Yaskawa INFORM job: OK_R2_O6-7(-90,0)OKKR.JBI

/JOB
//NAME OK_R2_O6-7(-90,0)OKKR
///FOLDERNAME X4
//POS
///NPOS 133,133,131,6,0,0
///TOOL 0
///POSTYPE PULSE
///PULSE
C00000=60285,-10095,-87170,10907,88181,-3199
C00001=89581,-19308,-95624,3409,86568,14234
C00002=122268,-16957,-60346,12820,63530,51265
C00003=120644,-15828,-53256,21467,67230,40646
C00004=120644,-14098,-51953,21456,67311,40660
C00005=120643,-14518,-52071,21476,67179,40636
C00006=120643,-15104,-51195,21601,66394,40485
C00007=120642,-17255,-54944,21425,67517,40699
C00008=120642,-17255,-54944,21425,67517,40699
C00009=124252,-5529,-45197,19318,66732,41820
C00010=124248,-5319,-45028,19320,66737,41819
C00011=124218,-3848,-43837,19334,66766,41814
C00012=124229,-4373,-44263,19329,66756,41816
C00013=124229,-5024,-43316,19456,65890,41667
C00014=124282,-6279,-47079,19198,67460,41953
C00015=120646,-13302,-53858,21234,68787,40941
C00016=120646,-14762,-51940,21506,66983,40600
C00017=120646,-14720,-50898,21598,66406,40487
C00018=120830,-17522,-52800,21535,66110,40497
C00019=120651,-14728,-51994,21496,67029,40610
C00020=120646,-14787,-50945,21602,66406,40490
C00021=120646,-14870,-50970,21605,66385,40483
C00022=120646,-14919,-51008,21604,66373,40480
C00023=120646,-15018,-51986,21521,66887,40581
C00024=120646,-13567,-53912,21247,68691,40923
C00025=105915,-38442,-90635,28282,81378,38856
C00026=57484,-69477,-110718,42573,54444,32820
C00027=-3643,-76224,-106676,-19950,71810,-76872
C00028=36671,-135259,-121545,10452,42336,6075
C00029=153552,-182601,-115262,-69180,49813,-17515
C00030=130897,-39590,-67652,-38094,64357,-42352
C00031=133939,-4658,-36155,-42635,61093,-39682
C00032=121252,36500,14973,-37087,50890,-41500
C00033=120918,45177,26978,-38391,48402,-40561
C00034=121382,52420,34740,-38113,53329,-33841
C00035=121382,52654,36258,-38487,52687,-33558
C00036=121382,52420,34740,-38113,53329,-33841
C00037=121377,54820,37402,-38294,53006,-33703
C00038=121382,52420,34740,-38113,53329,-33841
C00039=121917,44386,26656,-39102,48682,-40133
C00040=134879,58255,40786,-46614,53825,-35408
C00041=134959,60833,45092,-47358,52948,-34841
C00042=134959,61144,46552,-47770,52438,-34533
C00043=134959,60875,45298,-47416,52875,-34797
C00044=134857,63056,47803,-47604,52533,-34650
C00045=134959,60875,45298,-47416,52875,-34797
C00046=132891,53596,35323,-45210,53491,-36376
C00047=128554,62524,39730,-40860,62650,-37664
C00048=124660,52481,28282,-31369,57719,-36489
C00049=124396,62029,43751,-32872,53681,-35247
C00050=124397,61721,41951,-32506,54487,-35529
C00051=124441,58589,39965,-32677,54175,-35400
C00052=133765,73788,57651,-38360,55527,-31292
C00053=134326,62719,39703,-36596,60072,-32844
C00054=135410,51148,31829,-38776,48591,-44747
C00055=138156,57586,38014,-40647,49456,-43620
C00056=137577,66731,52697,-42929,45898,-42064
C00057=133639,60157,45125,-39794,45011,-44001
C00058=132456,59443,46653,-39908,43454,-43903
C00059=132752,49719,31225,-37339,47144,-45563
C00060=132976,-10381,-34918,-42251,48570,-38774
C00061=134698,-65118,-78640,-42103,61094,-39224
C00062=147917,-167168,-112708,-64264,48960,-21968
C00063=119754,-187210,-115895,-71836,42621,-17929
C00064=119758,-186866,-115850,-71681,42673,-18021
C00065=53896,-172979,-113746,-63904,34565,-25257
C00066=23682,-170517,-113316,-58323,27834,-29716
C00067=-3643,-76224,-106676,-19950,71810,-76872
C00068=64381,-28256,-98450,-10969,86693,-48952
C00069=88971,-14667,-95667,-7498,68279,-41414
C00070=119588,-13110,-62704,-15013,73832,-42943
C00071=119588,-13110,-62704,-15013,73832,-42943
C00072=120558,-12095,-59649,-15670,72677,-42495
C00073=120559,-10147,-58145,-15666,72751,-42503
C00074=120558,-10769,-58628,-15667,72729,-42501
C00075=120558,-10769,-58628,-15667,72729,-42501
C00076=120558,-11635,-57914,-15738,71876,-42387
C00077=120555,-12891,-60896,-15641,73024,-42540
C00078=95040,4780,-47974,-473,71962,-50162
C00079=96326,6971,-43876,-1258,70580,-49764
C00080=96504,8188,-42807,-1365,70550,-49710
C00081=96432,7698,-43239,-1322,70563,-49732
C00082=96432,6895,-42576,-1327,69744,-49725
C00083=96090,5943,-45717,-1110,71182,-49845
C00084=120646,-13948,-53489,-21604,68017,-40999
C00085=120646,-15353,-51537,-21891,66225,-40651
C00086=120646,-15164,-50572,-21969,65764,-40561
C00087=120651,-15325,-51597,-21886,66274,-40659
C00088=120458,-18091,-52377,-21925,65351,-40547
C00089=120646,-15383,-50573,-21989,65664,-40541
C00090=120646,-15549,-50757,-21980,65686,-40545
C00091=120646,-15089,-51509,-21872,66335,-40673
C00092=120646,-13673,-53452,-21587,68128,-41020
C00093=109799,-58506,-103025,-1655,56640,-68945
C00094=72582,-82093,-114007,4014,51361,-71324
C00095=52067,-53786,-27019,64889,38361,-39682
C00096=120741,-100002,-85602,9981,27010,44029
C00097=119621,-44404,-59771,8419,41423,45013
C00098=117663,-2811,-38597,8399,52217,45191
C00099=120702,21452,-13699,5381,57938,46744
C00100=116335,56883,35867,37385,59322,29596
C00101=116196,48699,28248,37279,59768,29706
C00102=116239,51251,31028,37399,59426,29593
C00103=116211,49643,29272,37323,59642,29665
C00104=116211,49822,31006,37666,58859,29354
C00105=116172,47372,26030,37059,60326,29912
C00106=106186,56602,32458,40868,65398,27238
C00107=106572,58996,37080,41208,63985,26816
C00108=106692,61436,39855,41307,63581,26700
C00109=106591,59390,37526,41224,63919,26799
C00110=106591,59599,39424,41561,63110,26445
C00111=106493,57459,35257,41134,64272,26904
C00112=115846,42546,19421,36690,61750,30302
C00113=117555,46608,31297,40428,52454,27269
C00114=120687,94317,83744,31652,39524,45736
C00115=120569,90994,80772,31662,39672,45727
C00116=110051,72582,62222,48229,50609,21848
C00117=111679,66904,55317,43745,47468,25399
C00118=112458,62952,41455,33837,55853,32000
C00119=111893,69063,52340,37068,50562,29781
C00120=111570,73580,54354,35260,54156,30929
C00121=111490,70901,52297,35345,54097,30866
C00122=107052,75469,60535,41045,50946,27156
C00123=107111,76128,56911,37464,55825,29367
C00124=111954,67372,45051,34070,56101,31848
C00125=111993,73411,55309,35316,53423,30857
C00126=113179,72507,56659,35287,51867,30842
C00127=112397,61419,38958,33599,56505,32200
C00128=120702,23915,-11347,5391,57756,46734
C00129=120707,-6637,-31564,7607,37304,45295
C00130=120737,-64904,-74687,7327,38208,45433
C00131=93974,-150495,-124706,8327,75713,42563
C00132=8894,-114644,-114160,10000,88881,39323
BC00000=260410,492998,972848
BC00001=270030,483686,999233
BC00002=258993,456898,1075139
BC00003=256299,434832,1075139
BC00004=256299,434832,1075139
BC00005=256299,434832,1075139
BC00006=256299,434832,1075139
BC00007=256299,434832,1075139
BC00008=203965,434832,1075139
BC00009=203965,434832,1075139
BC00010=203965,434832,1075139
BC00011=203965,434832,1075139
BC00012=203965,434832,1075139
BC00013=203965,434832,1075139
BC00014=203965,434832,1075139
BC00015=255837,442462,1075139
BC00016=256167,437012,1075139
BC00017=256299,434832,1075139
BC00018=256299,434832,1075139
BC00019=256299,434832,1075139
BC00020=251596,434014,1075139
BC00021=199069,424971,1075139
BC00022=194363,424171,1075139
BC00023=194231,426350,1075139
BC00024=193901,431800,1075139
BC00025=193901,431800,1075139
BC00026=193901,502169,1075139
BC00027=199448,515539,1075137
BC00028=185032,493226,660827
BC00029=170886,507346,17
BC00030=170886,499137,17
BC00031=170886,500820,17
BC00032=170886,503207,17
BC00033=170886,506149,17
BC00034=170886,504467,17
BC00035=170886,504467,17
BC00036=170886,504467,17
BC00037=170886,504467,17
BC00038=170886,504467,17
BC00039=170886,505099,17
BC00040=170886,505099,17
BC00041=170886,505099,17
BC00042=170886,505099,17
BC00043=170886,505099,17
BC00044=170886,505099,17
BC00045=170886,505099,17
BC00046=170886,505099,17
BC00047=183787,509866,15
BC00048=183787,509866,15
BC00049=183787,509866,15
BC00050=183787,509866,15
BC00051=183787,509866,15
BC00052=183787,509866,15
BC00053=183787,509866,15
BC00054=183787,509866,15
BC00055=183787,509866,15
BC00056=183787,509866,15
BC00057=183787,509866,15
BC00058=183787,509866,15
BC00059=183787,509866,15
BC00060=170886,507200,17
BC00061=170886,511894,17
BC00062=170886,502226,17
BC00063=170886,505869,17
BC00064=170886,506079,17
BC00065=170886,509232,17
BC00066=170886,502507,17
BC00067=199448,515539,1075137
BC00068=143041,501148,792030
BC00069=138642,496819,917141
BC00070=200892,451069,1075139
BC00071=195544,434280,1021239
BC00072=195544,434280,1021238
BC00073=195544,434280,1021238
BC00074=195544,434280,1021238
BC00075=195544,434280,1021238
BC00076=195544,434280,1021238
BC00077=195544,434280,1021238
BC00078=195544,434280,1021238
BC00079=195544,434280,1021238
BC00080=195544,434280,1021238
BC00081=195544,434280,1021238
BC00082=195544,434280,1021238
BC00083=195544,434280,1021238
BC00084=186560,442338,1075139
BC00085=186271,436877,1075139
BC00086=186156,434693,1075139
BC00087=186156,434693,1075139
BC00088=186156,434693,1075139
BC00089=243368,424735,1075139
BC00090=248072,423926,1075139
BC00091=248187,426110,1075139
BC00092=248476,431571,1075139
BC00093=248476,431571,1075139
BC00094=154886,508880,1075139
BC00095=226129,512135,483138
BC00096=268409,479745,74497
BC00097=268409,503413,53619
BC00098=268409,500913,17
BC00099=268409,507760,17
BC00100=268944,502290,17
BC00101=268944,493646,17
BC00102=268944,493646,17
BC00103=268944,493646,17
BC00104=268944,493646,17
BC00105=268944,493646,17
BC00106=268944,493646,17
BC00107=268944,493646,17
BC00108=268944,493646,17
BC00109=268944,493646,17
BC00110=268944,493646,17
BC00111=268944,493646,17
BC00112=268944,491895,17
BC00113=268943,496238,12
BC00114=254289,537584,17
BC00115=254289,537584,17
BC00116=268943,512909,14
BC00117=268944,512909,12
BC00118=268943,512909,14
BC00119=268943,512909,12
BC00120=268943,512909,12
BC00121=268943,512909,12
BC00122=268943,512909,14
BC00123=268943,512909,14
BC00124=268943,512909,14
BC00125=268943,512909,14
BC00126=268943,512909,14
BC00127=268943,512909,14
BC00128=268409,510422,17
BC00129=268409,508881,17
BC00130=268409,508951,17
BC00131=268409,511824,17
BC00132=268409,511683,17
EC00000=798297,-183828
EC00001=798261,-183829
EC00002=798156,-183832
EC00003=798156,-183832
EC00004=798156,-183832
EC00005=798156,-183832
EC00006=798156,-183832
EC00007=798156,-183832
EC00008=798156,-183832
EC00009=798156,-183832
EC00010=798156,-183832
EC00011=798156,-183832
EC00012=798156,-183832
EC00013=798156,-183832
EC00014=798156,-183832
EC00015=798156,-183832
EC00016=798156,-183832
EC00017=798156,-183832
EC00018=798156,-183832
EC00019=798156,-183832
EC00020=798156,-183832
EC00021=798156,-183832
EC00022=798156,-183832
EC00023=798156,-183832
EC00024=798156,-183832
EC00025=798156,-183832
EC00026=798156,-183832
EC00027=798156,-183832
EC00028=798156,-183832
EC00029=798156,-183832
EC00030=798156,-183832
EC00031=798156,-183832
EC00032=798156,-183832
EC00033=798156,-183832
EC00034=798156,-183832
EC00035=798156,-183832
EC00036=798156,-183832
EC00037=798156,-183832
EC00038=798156,-183832
EC00039=798156,-183832
EC00040=798156,-183832
EC00041=798156,-183832
EC00042=798156,-183832
EC00043=798156,-183832
EC00044=798156,-183832
EC00045=798156,-183832
EC00046=798156,-183832
EC00047=798154,-183831
EC00048=798154,-183831
EC00049=798154,-183831
EC00050=798154,-183831
EC00051=798154,-183831
EC00052=798154,-183831
EC00053=798154,-183831
EC00054=798154,-183831
EC00055=798154,-183831
EC00056=798154,-183831
EC00057=798154,-183831
EC00058=798154,-183831
EC00059=798154,-183831
EC00060=798156,-183832
EC00061=798156,-183832
EC00062=798156,-183832
EC00063=867082,-372677
EC00064=885768,-557346
EC00065=906795,-866627
EC00066=886351,-984978
EC00067=798156,-1296783
EC00068=798156,-1296783
EC00069=798156,-1296783
EC00070=798156,-1296783
EC00071=798156,-1296783
EC00072=798154,-1296783
EC00073=798154,-1296783
EC00074=798154,-1296783
EC00075=798154,-1296783
EC00076=798154,-1296783
EC00077=798154,-1296783
EC00078=798154,-1296783
EC00079=798154,-1296783
EC00080=798154,-1296783
EC00081=798154,-1296783
EC00082=798154,-1296783
EC00083=798154,-1296783
EC00084=798156,-1296783
EC00085=798156,-1296783
EC00086=798156,-1296783
EC00087=798156,-1296783
EC00088=798156,-1296783
EC00089=798156,-1296783
EC00090=798156,-1296783
EC00091=798156,-1296783
EC00092=798156,-1296783
EC00093=798156,-1296783
EC00094=798156,-1296783
EC00095=798156,-1296783
EC00096=798156,-1296783
EC00097=798156,-1296783
EC00098=798156,-1296783
EC00099=798156,-1296783
EC00100=798156,-1296783
EC00101=798156,-1296783
EC00102=798156,-1296783
EC00103=798156,-1296783
EC00104=798156,-1296783
EC00105=798156,-1296783
EC00106=798156,-1296783
EC00107=798156,-1296783
EC00108=798156,-1296783
EC00109=798156,-1296783
EC00110=798156,-1296783
EC00111=798156,-1296783
EC00112=798156,-1296783
EC00113=798154,-1296785
EC00114=798156,-1296783
EC00115=798156,-1296783
EC00116=798155,-1296784
EC00117=798154,-1296784
EC00118=798155,-1296784
EC00119=798154,-1296784
EC00120=798155,-1296784
EC00121=798155,-1296784
EC00122=798155,-1296784
EC00123=798155,-1296784
EC00124=798155,-1296784
EC00125=798155,-1296784
EC00126=798156,-1296783
EC00127=798156,-1296783
EC00128=798156,-1296783
EC00129=798156,-1296783
EC00130=798156,-1296783
///POSTYPE BASE
///RECTAN
///RCONF 0,0,0,0,1,0,0,0,0,0,0,0,0,0,0,0,0,0,0,0,0,0,0,0
P00006=2.006,1.622,-0.565,0.0000,0.0000,0.0000
P00021=0.073,2.058,-0.109,0.0000,0.0000,0.0000
P00022=2.006,1.622,-0.565,0.0000,0.0000,0.0000
///RCONF 0,0,0,0,0,0,0,0,0,0,0,0,0,0,0,0,0,0,0,0,0,0,0,0
P00023=-2.957,-4.083,2.762,0.0000,0.0000,0.0000
P00025=3.643,0.007,-2.585,0.0000,0.0000,0.0000
P00026=2.644,0.055,-2.583,0.0000,0.0000,0.0000
//INST
///DATE 2024/11/13 18:37
///ATTR SC,RW
///GROUP1 RB1,BS1
///GROUP2 ST1
NOP
'OK_r2_O6-7(-90,0)
'Spoina W6
'Path S1006
MOVJ C00000 BC00000 VJ=100.00  +MOVJ EC00000 VJ=10.00
MOVJ C00001 BC00001 VJ=100.00  +MOVJ EC00001 VJ=10.00
SFTOF3D
MOVJ C00002 BC00002 VJ=100.00  +MOVJ EC00002 VJ=100.00
SMOVL C00003 BC00003 V=100.0  +MOVJ EC00003
SREFP 3 C00004 BC00004  +REFP EC00004
CALL JOB:SEARCH-R1-S13D
SET P021 P006
SFTON3D P021
SMOVL C00005 BC00005 V=100.0  +MOVJ EC00005
SREFP 3 C00006 BC00006  +REFP EC00006
CALL JOB:SEARCH-R1-S13D
SET P021 P006
SFTON3D P021
SMOVL C00007 BC00007 V=100.0  +MOVJ EC00007
MOVL C00008 BC00008 V=400.0  +MOVJ EC00008 VJ=100.00
MOVL C00009 BC00009 V=400.0  +MOVJ EC00009 VJ=100.00
SMOVL C00010 BC00010 V=100.0  +MOVJ EC00010
SREFP 3 C00011 BC00011  +REFP EC00011
CALL JOB:SEARCH-R1-S13D
SET P022 P006
SFTON3D P022
SMOVL C00012 BC00012 V=100.0  +MOVJ EC00012
SREFP 3 C00013 BC00013  +REFP EC00013
CALL JOB:SEARCH-R1-S13D
SET P022 P006
SFTON3D P022
SMOVL C00014 BC00014 V=100.0  +MOVJ EC00014
'Path W937
SFTOF3D
MOVJ C00015 BC00015 VJ=50.00  +MOVJ EC00015 VJ=100.00
SMOVL C00016 BC00016 V=400.0  +MOVJ EC00016
SFTON3D P021
SMOVL C00017 BC00017 V=100.0 PL=0  +MOVJ EC00017
SREFP 1 C00018 BC00018  +REFP EC00018
SREFP 2 C00019 BC00019  +REFP EC00019
MACRO1 MJ#(0) ARGF6
ARCON
SMOVL C00020 BC00020 V=8.3  +MOVJ EC00020
SFTON3D P022
SMOVL C00021 BC00021 V=8.3  +MOVJ EC00021
SMOVL C00022 BC00022 V=8.3  +MOVJ EC00022
ARCOF
SMOVL C00023 BC00023 V=400.0  +MOVJ EC00023
SFTOF3D
SMOVL C00024 BC00024 V=1000.0  +MOVJ EC00024
MOVJ C00025 BC00025 VJ=100.00  +MOVJ EC00025 VJ=10.00
MOVJ C00026 BC00026 VJ=100.00  +MOVJ EC00026 VJ=100.00
MOVJ C00027 BC00027 VJ=100.00  +MOVJ EC00027 VJ=100.00
SFTOF3D
CALL JOB:CLEAN-R1_KM_NEW
'wire_cut
SFTOF
'wire_cut
MOVJ C00028 BC00028 VJ=100.00  +MOVJ EC00028 VJ=100.00
MOVJ C00029 BC00029 VJ=100.00  +MOVJ EC00029 VJ=100.00
MOVJ C00030 BC00030 VJ=50.00  +MOVJ EC00030 VJ=100.00
MOVJ C00031 BC00031 VJ=50.00  +MOVJ EC00031 VJ=100.00
'Path S1300
SFTOF3D
MOVJ C00032 BC00032 VJ=50.00  +MOVJ EC00032 VJ=100.00
MOVL C00033 BC00033 V=100.0  +MOVJ EC00033 VJ=100.00
SMOVL C00034 BC00034 V=100.0  +MOVJ EC00034
SREFP 3 C00035 BC00035  +REFP EC00035
CALL JOB:SEARCH-R1-S13D
SET P025 P006
SFTON3D P025
SMOVL C00036 BC00036 V=100.0  +MOVJ EC00036
SREFP 3 C00037 BC00037  +REFP EC00037
CALL JOB:SEARCH-R1-S13D
SET P025 P006
SFTON3D P025
SMOVL C00038 BC00038 V=100.0  +MOVJ EC00038
MOVL C00039 BC00039 V=400.0  +MOVJ EC00039 VJ=100.00
SMOVL C00040 BC00040 V=400.0  +MOVJ EC00040
SMOVL C00041 BC00041 V=100.0  +MOVJ EC00041
SREFP 3 C00042 BC00042  +REFP EC00042
CALL JOB:SEARCH-R1-S13D
SET P026 P006
SFTON3D P026
SMOVL C00043 BC00043 V=100.0  +MOVJ EC00043
SREFP 3 C00044 BC00044  +REFP EC00044
CALL JOB:SEARCH-R1-S13D
SET P026 P006
SFTON3D P026
SMOVL C00045 BC00045 V=100.0  +MOVJ EC00045
MOVL C00046 BC00046 V=1000.0  +MOVJ EC00046 VJ=100.00
'Path W1301
SFTOF3D
SFTON3D P025
MOVJ C00047 BC00047 VJ=50.00  +MOVJ EC00047 VJ=100.00
SMOVL C00048 BC00048 V=400.0  +MOVJ EC00048
SFTON3D P025
SMOVL C00049 BC00049 V=100.0 PL=0  +MOVJ EC00049
SREFP 1 C00050 BC00050  +REFP EC00050
SREFP 2 C00051 BC00051  +REFP EC00051
MACRO1 MJ#(0) ARGF6
ARCON
SWVON WEV#(30)
SMOVL C00052 BC00052 V=8.3  +MOVJ EC00052
ARCOF
SWVOF
MOVJ C00053 BC00053 VJ=50.00  +MOVJ EC00053 VJ=10.00
SFTOF3D
MOVJ C00054 BC00054 VJ=50.00  +MOVJ EC00054 VJ=10.00
MOVJ C00055 BC00055 VJ=50.00  +MOVJ EC00055 VJ=10.00
MACRO1 MJ#(0) ARGF6
SFTON3D P026
SMOVL C00056 BC00056 V=100.0  +MOVJ EC00056
ARCON
SWVON WEV#(30)
ARCON
SMOVL C00057 BC00057 V=7.5  +MOVJ EC00057
SMOVL C00058 BC00058 V=10.0  +MOVJ EC00058
ARCOF
SWVOF
MOVJ C00059 BC00059 VJ=100.00  +MOVJ EC00059 VJ=10.00
SFTOF3D
MOVJ C00060 BC00060 VJ=100.00  +MOVJ EC00060 VJ=100.00
MOVJ C00061 BC00061 VJ=100.00  +MOVJ EC00061 VJ=100.00
'OBROT_SPRAWDZIC
MOVJ C00062 BC00062 VJ=100.00  +MOVJ EC00062 VJ=100.00
MOVJ C00063 BC00063 VJ=100.00  +MOVJ EC00063 VJ=100.00
MOVJ C00064 BC00064 VJ=100.00  +MOVJ EC00064 VJ=100.00
MOVJ C00065 BC00065 VJ=100.00  +MOVJ EC00065 VJ=100.00
MOVJ C00066 BC00066 VJ=100.00  +MOVJ EC00066 VJ=100.00
MOVJ C00067 BC00067 VJ=100.00  +MOVJ EC00067 VJ=100.00
CALL JOB:CLEAN-R1_KM_NEW
'wire_cut
'wire_cut
'Path S1296
MOVJ C00068 BC00068 VJ=100.00  +MOVJ EC00068 VJ=10.00
MOVJ C00069 BC00069 VJ=100.00  +MOVJ EC00069 VJ=10.00
SFTOF3D
MOVJ C00070 BC00070 VJ=100.00  +MOVJ EC00070 VJ=100.00
MOVL C00071 BC00071 V=100.0  +MOVJ EC00071 VJ=100.00
SMOVL C00072 BC00072 V=100.0  +MOVJ EC00072
SREFP 3 C00073 BC00073  +REFP EC00073
CALL JOB:SEARCH-R1-S13D
SET P021 P006
SFTON3D P021
SMOVL C00074 BC00074 V=100.0  +MOVJ EC00074
SMOVL C00075 BC00075 V=100.0  +MOVJ EC00075
SREFP 3 C00076 BC00076  +REFP EC00076
CALL JOB:SEARCH-R1-S13D
SET P021 P006
SFTON3D P021
SFTOF3D
SMOVL C00077 BC00077 V=100.0  +MOVJ EC00077
MOVJ C00078 BC00078 VJ=50.00  +MOVJ EC00078 VJ=50.00
'POMIAR 2
SMOVL C00079 BC00079 V=100.0  +MOVJ EC00079
SREFP 3 C00080 BC00080  +REFP EC00080
CALL JOB:SEARCH-R1-S13D
SET P022 P006
SFTON3D P022
SMOVL C00081 BC00081 V=100.0  +MOVJ EC00081
SREFP 3 C00082 BC00082  +REFP EC00082
CALL JOB:SEARCH-R1-S13D
SET P022 P006
SFTON3D P022
SMOVL C00083 BC00083 V=100.0  +MOVJ EC00083
'Path W1297
SFTOF3D
SFTON3D P021
MOVJ C00084 BC00084 VJ=50.00  +MOVJ EC00084 VJ=100.00
SMOVL C00085 BC00085 V=400.0  +MOVJ EC00085
SMOVL C00086 BC00086 V=100.0 PL=0  +MOVJ EC00086
SREFP 1 C00087 BC00087  +REFP EC00087
SREFP 2 C00088 BC00088  +REFP EC00088
MACRO1 MJ#(0) ARGF6
ARCON
SMOVL C00089 BC00089 V=9.2  +MOVJ EC00089
SMOVL C00090 BC00090 V=9.2  +MOVJ EC00090
ARCOF
SWVOF
SMOVL C00091 BC00091 V=400.0  +MOVJ EC00091
SMOVL C00092 BC00092 V=1000.0  +MOVJ EC00092
MOVJ C00093 BC00093 VJ=100.00  +MOVJ EC00093 VJ=10.00
MOVJ C00094 BC00094 VJ=100.00  +MOVJ EC00094 VJ=10.00
SFTOF3D
CALL JOB:CLEAN-R1_KM_NEW
'wire_cut
'wire_cut
'Spoina W7
MOVJ C00095 BC00095 VJ=100.00  +MOVJ EC00095 VJ=10.00
MOVJ C00096 BC00096 VJ=100.00  +MOVJ EC00096 VJ=100.00
MOVJ C00097 BC00097 VJ=100.00  +MOVJ EC00097 VJ=50.00
MOVJ C00098 BC00098 VJ=100.00  +MOVJ EC00098 VJ=10.00
MOVJ C00099 BC00099 VJ=100.00  +MOVJ EC00099 VJ=100.00
'Path S1298
SFTOF3D
MOVL C00100 BC00100 V=400.0  +MOVJ EC00100 VJ=100.00
SMOVL C00101 BC00101 V=100.0  +MOVJ EC00101
SREFP 3 C00102 BC00102  +REFP EC00102
CALL JOB:SEARCH-R1-S13D
SET P023 P006
SFTON3D P023
SMOVL C00103 BC00103 V=100.0  +MOVJ EC00103
SREFP 3 C00104 BC00104  +REFP EC00104
CALL JOB:SEARCH-R1-S13D
SET P023 P006
SFTON3D P023
SFTOF3D
SMOVL C00105 BC00105 V=100.0  +MOVJ EC00105
'POMIAR 2
MOVJ C00106 BC00106 VJ=50.00  +MOVJ EC00106 VJ=50.00
SMOVL C00107 BC00107 V=100.0  +MOVJ EC00107
SREFP 3 C00108 BC00108  +REFP EC00108
CALL JOB:SEARCH-R1-S13D
SET P021 P006
SFTON3D P021
SMOVL C00109 BC00109 V=100.0  +MOVJ EC00109
SREFP 3 C00110 BC00110  +REFP EC00110
CALL JOB:SEARCH-R1-S13D
SET P021 P006
SFTON3D P021
SMOVL C00111 BC00111 V=166.7  +MOVJ EC00111
MOVL C00112 BC00112 V=400.0  +MOVJ EC00112 VJ=100.00
'Path W1299
SFTOF3D
SFTON3D P023
SMOVL C00113 BC00113 V=100.0 PL=0  +MOVJ EC00113
SREFP 1 C00114 BC00114  +REFP EC00114
SREFP 2 C00115 BC00115  +REFP EC00115
MACRO1 MJ#(0) ARGF14
ARCON
SWVON WEV#(30)
SMOVL C00116 BC00116 V=9.2  +MOVJ EC00116
SMOVL C00117 BC00117 V=9.2  +MOVJ EC00117
ARCOF
SWVOF
MOVJ C00118 BC00118 VJ=100.00  +MOVJ EC00118 VJ=10.00
SFTON3D P021
SMOVL C00119 BC00119 V=100.0 PL=0  +MOVJ EC00119
REFP 1 RB1 C00120 BC00120
REFP 2 RB1 C00121 BC00121
ARCON
SWVON WEV#(30)
SMOVL C00122 BC00122 V=7.5  +MOVJ EC00120
ARCOF
SWVOF
MOVJ C00123 BC00123 VJ=50.00  +MOVJ EC00121 VJ=10.00
MOVJ C00124 BC00124 VJ=50.00  +MOVJ EC00122 VJ=10.00
SMOVL C00125 BC00125 V=33.3 PL=0  +MOVJ EC00123
ARCON
SMOVL C00126 BC00126 V=13.3  +MOVJ EC00124
ARCOF
MOVJ C00127 BC00127 VJ=100.00  +MOVJ EC00125 VJ=10.00
SFTOF3D
MOVJ C00128 BC00128 VJ=100.00  +MOVJ EC00126 VJ=100.00
MOVJ C00129 BC00129 VJ=100.00  +MOVJ EC00127 VJ=10.00
MOVJ C00130 BC00130 VJ=100.00  +MOVJ EC00128 VJ=100.00
MOVJ C00131 BC00131 VJ=100.00  +MOVJ EC00129 VJ=10.00
MOVJ C00132 BC00132 VJ=100.00  +MOVJ EC00130 VJ=10.00
END
